DEVICE_TYPE RMT_DEV (* Remotely Managed Device Type *)
  (* Standard: 61499 ITA; Description: Remotely Managed Device *)
  (* Version 0.4, 2007-10-10, JHC, Holobloc Inc, Moved to fb.rt. *)
  (* Version 0.3, 2000-12-22, JHC, Rockwell Automation, Back to no DM_RES *)
  (* Version 0.2, 2000-12-20, JHC, Rockwell Automation, Now contains DM_RES *)
  (* Version 0.1, 2000-05-16, JHC, Rockwell Automation, File type changed to ".dev" *)
  (* Version 0.0, 2000-03-19, JHC, Rockwell Automation *)
  (* Compiler header: package fb.rt; *)
  (* Compiler classdef: public class RMT_DEV extends FBDevice implements RemoteDevice *)
  (* Compiler Java IBM VisualAge 3.0 *)
  VAR_INPUT
    MGR_ID : WSTRING := "localhost:61499"; (* Device manager socket ID *)
  END_VAR
  RESOURCE MGR : RMT_RES
  END_RESOURCE
  DATA_CONNECTIONS
    MGR_ID TO MGR.MGR_ID;
  END_CONNECTIONS
END_DEVICE_TYPE
